# EPICS StreamDevice protocol: cognexDataMan100/dataman.proto
Terminator = CR;
ReadTimeout = 1000;

read {
    in "%s";
}
